// TIA Portal project "Practice" (V18)

(* hardware
DEVICE "S7-1500/ET200MP station_1"  S7-1500 station
   slot 0: "Rail_0"  Rack  6ES7 590-1***0-0AA0
   slot 1: "PLC_1"  CPU 1516F-3 PN/DP  6ES7 516-3FN01-0AB0  V2.1
      slot 3: "CPU display_1"  6ES7591-1BA00-0AA0
      slot 32768: "PROFINET interface_1"  X1
         slot 32769: "Port_1"  X1 P1
         slot 32770: "Port_2"  X1 P2
      slot 33024: "PROFINET interface_2"  X2
         slot 33025: "Port_1"  X2 P1
      slot 33280: "DP interface_1"  X3
   slot 2: "DI 16x24VDC HF_1"  DI 16x24VDC HF  6ES7 521-1BH00-0AB0  V2.2
   slot 3: "DQ 16x24VDC/0.5A HF_1"  DQ 16x24VDC/0.5A HF  6ES7 522-1BH01-0AB0  V1.1
   slot 4: "AI 8xU/I HF_1"  AI 8xU/I HF  6ES7 531-7NF00-0AB0  V1.2
   slot 5: "AQ 4xU/I HF_1"  AQ 4xU/I HF  6ES7 532-5ND00-0AB0  V1.1
*)

// ===== PLC "PLC_1"  CPU 1516F-3 PN/DP =====

VAR_GLOBAL   // PLC tag table "Default tag table"
   "ON" AT %I0.0 : Bool;
   "OFF" AT %I0.1 : Bool;
   "LAMP" AT %Q0.0 : Bool;
   "FAN" AT %Q0.1 : Bool;
   "WAR_LAMP" AT %Q0.2 : Bool;
   "CH_LP" AT %Q0.3 : Bool;
   "RST" AT %I0.2 : Bool;
   "POW_ON" AT %I0.3 : Bool;
   "CH_RST" AT %I0.4 : Bool;
   "CH_LAMP" AT %I0.5 : Bool;
END_VAR

DATA_BLOCK "Main_Safety_RTG1_DB"   // DB1, F_DB
{ S7_Optimized_Access := 'TRUE' }
NAME : FUSI
VERSION : 0.1
// stored: InstanceOfName Main_Safety_RTG1
"Main_Safety_RTG1"
BEGIN
END_DATA_BLOCK

DATA_BLOCK "SELF_HOLDING01_FB_DB"   // DB2
{ S7_Optimized_Access := 'TRUE' }
VERSION : 0.1
// stored: InstanceOfName SELF_HOLDING01_FB
"SELF_HOLDING01_FB"
BEGIN
END_DATA_BLOCK

DATA_BLOCK "SELF_HOLD_TIMER_FB02_DB"   // DB3
{ S7_Optimized_Access := 'TRUE' }
VERSION : 0.1
// stored: InstanceOfName SELF_HOLD_TIMER_FB02
"SELF_HOLD_TIMER_FB02"
BEGIN
END_DATA_BLOCK

DATA_BLOCK "SELF_HOLD_TOFF_FB03_DB"   // DB4
{ S7_Optimized_Access := 'TRUE' }
VERSION : 0.1
// stored: InstanceOfName SELF_HOLD_TOFF_FB03
"SELF_HOLD_TOFF_FB03"
BEGIN
END_DATA_BLOCK

DATA_BLOCK "LAMP_FAN_FLK_FB05_DB"   // DB5
{ S7_Optimized_Access := 'TRUE' }
VERSION : 0.1
// stored: InstanceOfName LAMP_FAN_FLK_FB05
"LAMP_FAN_FLK_FB05"
BEGIN
END_DATA_BLOCK

DATA_BLOCK "SELF_HOLD_RETENTIV_FB07_DB"   // DB6
{ S7_Optimized_Access := 'TRUE' }
VERSION : 0.1
// stored: InstanceOfName SELF_HOLD_RETENTIV_FB07
"SELF_HOLD_RETENTIV_FB07"
BEGIN
END_DATA_BLOCK

DATA_BLOCK "TOT_FUN_FB09_DB"   // DB7
{ S7_Optimized_Access := 'TRUE' }
VERSION : 0.1
// stored: InstanceOfName TOT_FUN_FB09
"TOT_FUN_FB09"
BEGIN
END_DATA_BLOCK

FUNCTION_BLOCK "Main_Safety_RTG1"   // FB1, F_FBD
{ S7_Optimized_Access := 'TRUE' }
BEGIN
END_FUNCTION_BLOCK

FUNCTION_BLOCK "SELF_HOLDING01_FB"   // FB2, LAD
TITLE = 자기유지 회로를 사용하여 램프 점등하기
{ S7_Optimized_Access := 'TRUE' }
VERSION : 0.1
   VAR_INPUT
      ON : Bool;
      OFF : Bool;
   END_VAR
   VAR_OUTPUT
      LAMP : Bool;
   END_VAR
   VAR
      K1 : Bool;
   END_VAR
BEGIN

REGION Network 1: 램프 점등을 위한 자기유지회로
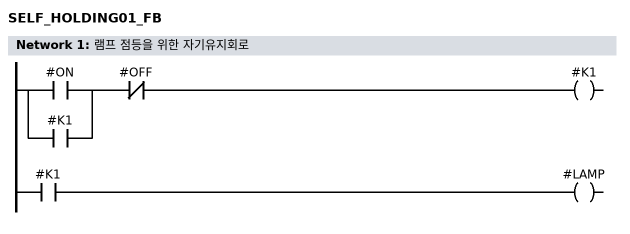
   RUNG wire#powerrail
      Contact( #ON )
      wire#w1
      I_Contact( #OFF )
      Coil( #K1 )
   END_RUNG
   RUNG wire#powerrail
      Contact( #K1 )
   END_RUNG wire#w1
   RUNG wire#powerrail
      Contact( #K1 )
      Coil( #LAMP )
   END_RUNG
   // the same network as SCL:
   #K1 := (#ON OR #K1) AND NOT #OFF;
   #LAMP := #K1;
END_REGION
END_FUNCTION_BLOCK

FUNCTION_BLOCK "SELF_HOLD_TIMER_FB02"   // FB3, LAD
TITLE = 자기유지 회로와 타이머의 조합 1
{ S7_Optimized_Access := 'TRUE' }
VERSION : 0.1
   VAR_INPUT
      ON : Bool;
      OFF : Bool;
   END_VAR
   VAR_OUTPUT
      LAMP : Bool;
      FAN : Bool;
   END_VAR
   VAR
      K1 : Bool;
      K2 : Bool;
      T1_Q : Bool;
      IEC_Timer_0_Instance : TON_TIME;
   END_VAR
BEGIN

REGION Network 1: 램프 제어 자기유지회로
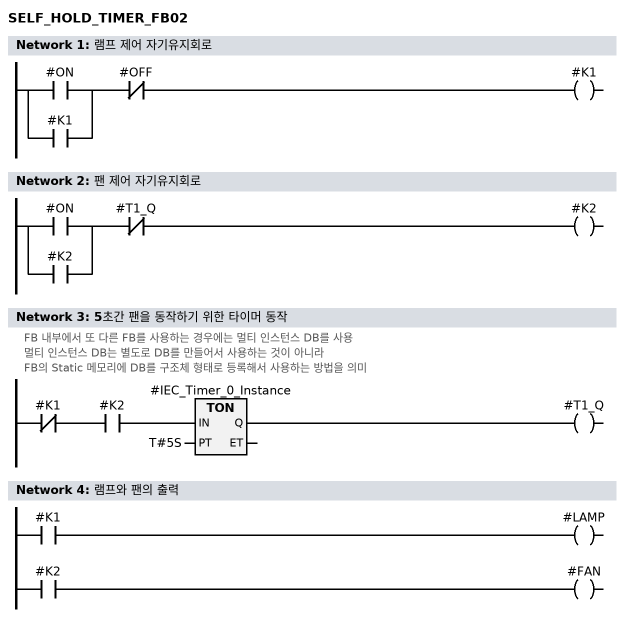
   RUNG wire#powerrail
      Contact( #ON )
      wire#w1
      I_Contact( #OFF )
      Coil( #K1 )
   END_RUNG
   RUNG wire#powerrail
      Contact( #K1 )
   END_RUNG wire#w1
   // the same network as SCL:
   #K1 := (#ON OR #K1) AND NOT #OFF;
END_REGION

REGION Network 2: 팬 제어 자기유지회로
   RUNG wire#powerrail
      Contact( #ON )
      wire#w1
      I_Contact( #T1_Q )
      Coil( #K2 )
   END_RUNG
   RUNG wire#powerrail
      Contact( #K2 )
   END_RUNG wire#w1
   // the same network as SCL:
   #K2 := (#ON OR #K2) AND NOT #T1_Q;
END_REGION

REGION Network 3: 5초간 팬을 동작하기 위한 타이머 동작
   // FB 내부에서 또 다른 FB를 사용하는 경우에는 멀티 인스턴스 DB를 사용
   // 
   // 멀티 인스턴스 DB는 별도로 DB를 만들어서 사용하는 것이 아니라
   // FB의 Static 메모리에 DB를 구조체 형태로 등록해서 사용하는 방법을 의미
   #IEC_Timer_0_Instance(IN := NOT #K1 AND #K2, PT := T#5S);   // TON
   #T1_Q := #IEC_Timer_0_Instance.Q;
END_REGION

REGION Network 4: 램프와 팬의 출력
   RUNG wire#powerrail
      Contact( #K1 )
      Coil( #LAMP )
   END_RUNG
   RUNG wire#powerrail
      Contact( #K2 )
      Coil( #FAN )
   END_RUNG
   // the same network as SCL:
   #LAMP := #K1;
   #FAN := #K2;
END_REGION
END_FUNCTION_BLOCK

FUNCTION_BLOCK "SELF_HOLD_TOFF_FB03"   // FB4, LAD
TITLE = 자기유지 회로와 타이머의 조합 2
{ S7_Optimized_Access := 'TRUE' }
VERSION : 0.1
   VAR_INPUT
      ON : Bool;
      OFF : Bool;
   END_VAR
   VAR_OUTPUT
      LAMP : Bool;
      FAN : Bool;
   END_VAR
   VAR
      K1 : Bool;
      K2 : Bool;
      IEC_Timer_0_Instance : TOF_TIME;
   END_VAR
BEGIN

REGION Network 1: 램프 제어 자기유지회로
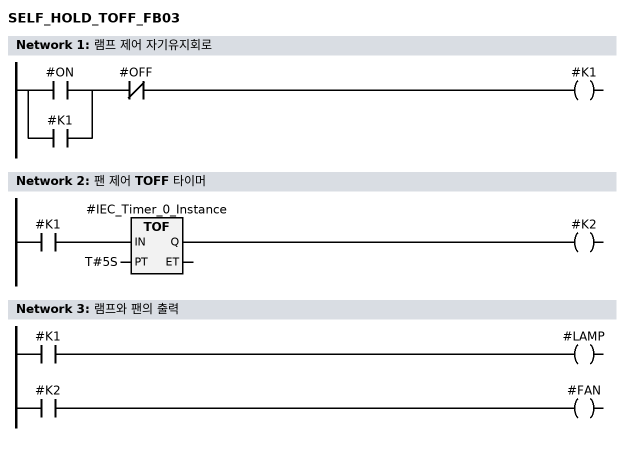
   RUNG wire#powerrail
      Contact( #ON )
      wire#w1
      I_Contact( #OFF )
      Coil( #K1 )
   END_RUNG
   RUNG wire#powerrail
      Contact( #K1 )
   END_RUNG wire#w1
   // the same network as SCL:
   #K1 := (#ON OR #K1) AND NOT #OFF;
END_REGION

REGION Network 2: 팬 제어 TOFF 타이머
   #IEC_Timer_0_Instance(IN := #K1, PT := T#5S);   // TOF
   #K2 := #IEC_Timer_0_Instance.Q;
END_REGION

REGION Network 3: 램프와 팬의 출력
   RUNG wire#powerrail
      Contact( #K1 )
      Coil( #LAMP )
   END_RUNG
   RUNG wire#powerrail
      Contact( #K2 )
      Coil( #FAN )
   END_RUNG
   // the same network as SCL:
   #LAMP := #K1;
   #FAN := #K2;
END_REGION
END_FUNCTION_BLOCK

FUNCTION_BLOCK "FLICKER_FB04"   // FB5, LAD
TITLE = 플리커 타이머 사용하기
{ S7_Optimized_Access := 'TRUE' }
VERSION : 0.1
   VAR_INPUT
      ON : Bool;
   END_VAR
   VAR_OUTPUT
      FLK_OUT : Bool;
   END_VAR
   VAR
      T1_Q : Bool;
      T1_ET : Time;
      IEC_Timer_0_Instance : TON_TIME;
   END_VAR
   VAR_TEMP   // added for the SCL form of the ladder/FBD networks
      _w1 : Bool;
   END_VAR
BEGIN

REGION Network 1: 1Hz주기를 가진 FLICKER 타이머
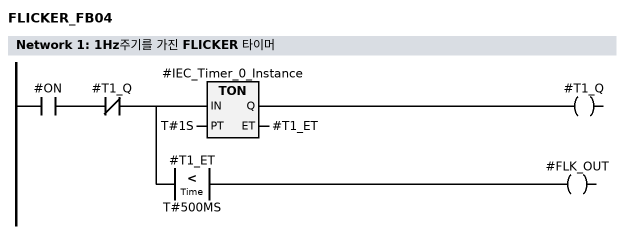
   #_w1 := #ON AND NOT #T1_Q;
   #IEC_Timer_0_Instance(IN := #_w1, PT := T#1S, ET => #T1_ET);   // TON
   #T1_Q := #IEC_Timer_0_Instance.Q;
   #FLK_OUT := #_w1 AND (#T1_ET < T#500MS);
END_REGION
END_FUNCTION_BLOCK

FUNCTION_BLOCK "LAMP_FAN_FLK_FB05"   // FB6, LAD
TITLE = 플리커 타이머 사용하기
{ S7_Optimized_Access := 'TRUE' }
VERSION : 0.1
   VAR_INPUT
      ON : Bool;
      OFF : Bool;
   END_VAR
   VAR_OUTPUT
      LAMP : Bool;
      FAN : Bool;
      WAR_LAMP : Bool;
   END_VAR
   VAR
      K1 : Bool;
      K2 : Bool;
      SELF_HOLD_TOFF_FB03_Instance : "SELF_HOLD_TOFF_FB03";
      FLICKER_FB04_Instance : "FLICKER_FB04";
   END_VAR
BEGIN

REGION Network 1: FB05에서 FB03 호출
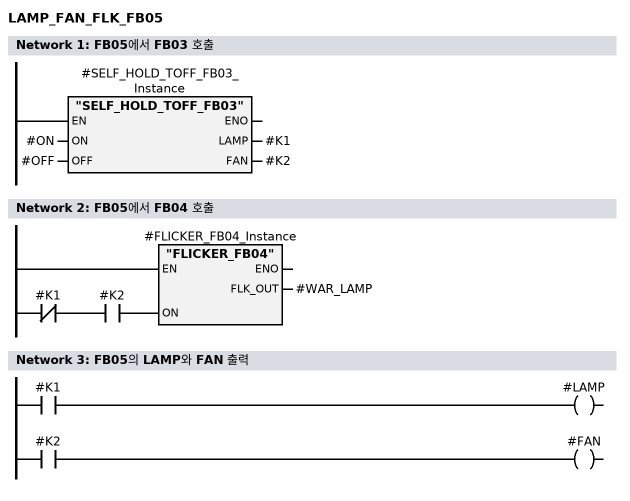
   RUNG wire#powerrail
      #SELF_HOLD_TOFF_FB03_Instance(ON := #ON, OFF := #OFF, LAMP => #K1, FAN => #K2)
   END_RUNG
   // the same network as SCL:
   #SELF_HOLD_TOFF_FB03_Instance(ON := #ON, OFF := #OFF, LAMP => #K1, FAN => #K2);   // "SELF_HOLD_TOFF_FB03"
END_REGION

REGION Network 2: FB05에서 FB04 호출
   RUNG wire#powerrail
      #FLICKER_FB04_Instance(ON := wire#w1, FLK_OUT => #WAR_LAMP)
   END_RUNG
   RUNG wire#powerrail
      I_Contact( #K1 )
      Contact( #K2 )
   END_RUNG wire#w1
   // the same network as SCL:
   #FLICKER_FB04_Instance(ON := NOT #K1 AND #K2, FLK_OUT => #WAR_LAMP);   // "FLICKER_FB04"
END_REGION

REGION Network 3: FB05의 LAMP와 FAN 출력
   RUNG wire#powerrail
      Contact( #K1 )
      Coil( #LAMP )
   END_RUNG
   RUNG wire#powerrail
      Contact( #K2 )
      Coil( #FAN )
   END_RUNG
   // the same network as SCL:
   #LAMP := #K1;
   #FAN := #K2;
END_REGION
END_FUNCTION_BLOCK

FUNCTION_BLOCK "RETENTIV_TIME_FB06"   // FB7, LAD
TITLE = PLC의 전원 ON/OFF에 관계없이 경과시간과 카운터의 값을 기억하기 위해서
{ S7_Optimized_Access := 'TRUE' }
VERSION : 0.1
   VAR_INPUT
      ON : Bool;
      RST : Bool;
   END_VAR
   VAR_OUTPUT
      OUT : Bool;
   END_VAR
   VAR
      T1_Q : Bool;
      C1_Q : Bool;
   END_VAR
   VAR RETAIN
      IEC_Timer_0_Instance : TONR_TIME;
      IEC_Counter_0_Instance : CTU_INT;
   END_VAR
BEGIN

REGION Network 1: 적산타이머의 동작
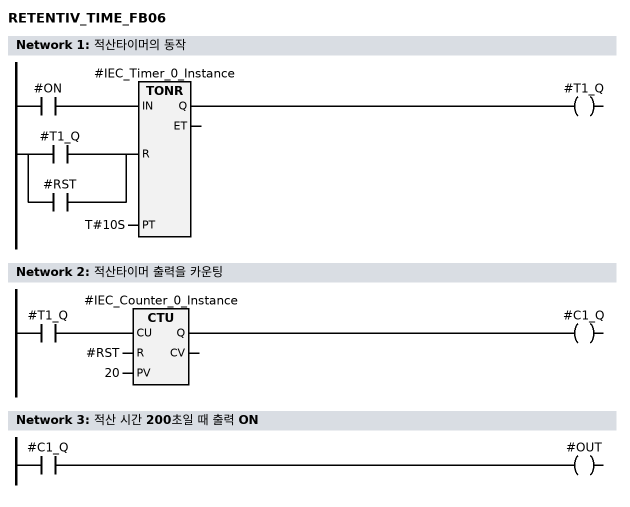
   #IEC_Timer_0_Instance(IN := #ON, R := #T1_Q OR #RST, PT := T#10S);   // TONR
   #T1_Q := #IEC_Timer_0_Instance.Q;
END_REGION

REGION Network 2: 적산타이머 출력을 카운팅
   #IEC_Counter_0_Instance(CU := #T1_Q, R := #RST, PV := 20);   // CTU
   #C1_Q := #IEC_Counter_0_Instance.Q;
END_REGION

REGION Network 3: 적산 시간 200초일 때 출력 ON
   RUNG wire#powerrail
      Contact( #C1_Q )
      Coil( #OUT )
   END_RUNG
   // the same network as SCL:
   #OUT := #C1_Q;
END_REGION
END_FUNCTION_BLOCK

FUNCTION_BLOCK "SELF_HOLD_RETENTIV_FB07"   // FB8, LAD
TITLE = FB1의 램프 출력은 FB6의 ON 입력으로 사용(K1 지정)
{ S7_Optimized_Access := 'TRUE' }
VERSION : 0.1
   VAR_INPUT
      ON : Bool;
      OFF : Bool;
      RST : Bool;
   END_VAR
   VAR_OUTPUT
      LAMP : Bool;
      CH_LP : Bool;
   END_VAR
   VAR
      K1 : Bool;
      SELF_HOLDING01_FB_Instance : "SELF_HOLDING01_FB";
      RETENTIV_TIME_FB06_Instance : "RETENTIV_TIME_FB06";
   END_VAR
BEGIN

REGION Network 1: 램프 점들을 위한 자기유지회로
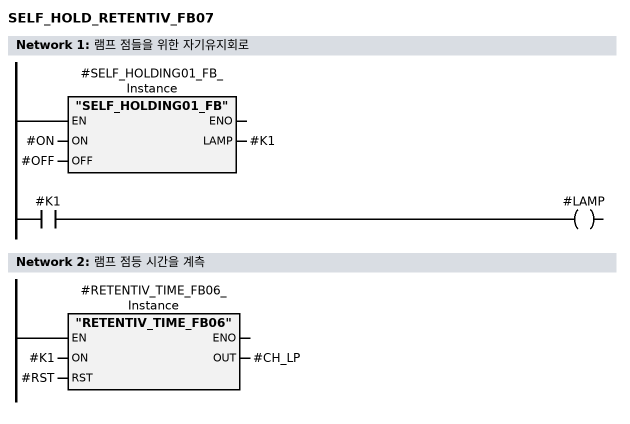
   RUNG wire#powerrail
      #SELF_HOLDING01_FB_Instance(ON := #ON, OFF := #OFF, LAMP => #K1)
   END_RUNG
   RUNG wire#powerrail
      Contact( #K1 )
      Coil( #LAMP )
   END_RUNG
   // the same network as SCL:
   #SELF_HOLDING01_FB_Instance(ON := #ON, OFF := #OFF, LAMP => #K1);   // "SELF_HOLDING01_FB"
   #LAMP := #K1;
END_REGION

REGION Network 2: 램프 점등 시간을 계측
   RUNG wire#powerrail
      #RETENTIV_TIME_FB06_Instance(ON := #K1, RST := #RST, OUT => #CH_LP)
   END_RUNG
   // the same network as SCL:
   #RETENTIV_TIME_FB06_Instance(ON := #K1, RST := #RST, OUT => #CH_LP);   // "RETENTIV_TIME_FB06"
END_REGION
END_FUNCTION_BLOCK

FUNCTION_BLOCK "FF_FUN_FB08"   // FB9, LAD
{ S7_Optimized_Access := 'TRUE' }
VERSION : 0.1
   VAR_INPUT
      ON_OFF : Bool;
      CH_RST : Bool;
   END_VAR
   VAR_OUTPUT
      ON_OUT : Bool;
      OFF_OUT : Bool;
      RST_OUT : Bool;
   END_VAR
   VAR
      K1 : Bool;
      K2 : Bool;
      R_EG01 : Bool;
      R_EG02 : Bool;
      F_EG01 : Bool;
      T1_Q : Bool;
      IEC_Timer_0_Instance : TON_TIME;
   END_VAR
BEGIN

REGION Network 1: 스위치 입력을 상승펄스 신호로 변경하여 K2를 토글 동작하도록 프로그램 작성
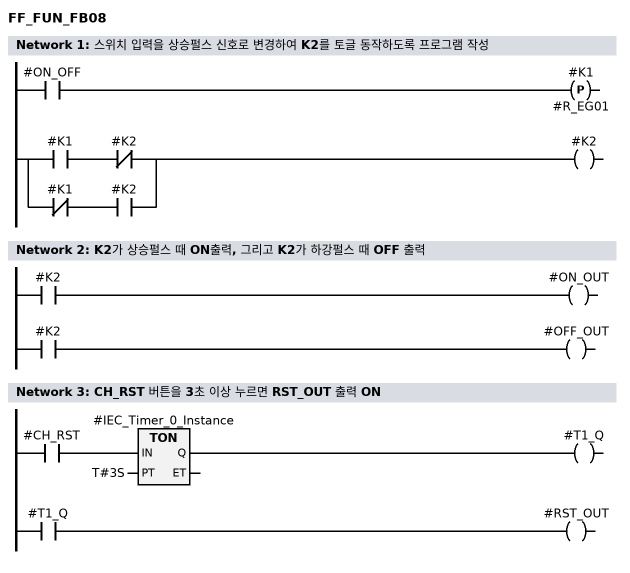
   #K1 := #ON_OFF AND NOT #R_EG01;   // rising edge
   #R_EG01 := #ON_OFF;
   #K2 := (#K1 AND NOT #K2) OR (NOT #K1 AND #K2);
END_REGION

REGION Network 2: K2가 상승펄스 때 ON출력, 그리고 K2가 하강펄스 때 OFF 출력
   RUNG wire#powerrail
      Contact( #K2 )
      Coil( #ON_OUT )
   END_RUNG
   RUNG wire#powerrail
      Contact( #K2 )
      Coil( #OFF_OUT )
   END_RUNG
   // the same network as SCL:
   #ON_OUT := #K2;
   #OFF_OUT := #K2;
END_REGION

REGION Network 3: CH_RST 버튼을 3초 이상 누르면 RST_OUT 출력 ON
   #IEC_Timer_0_Instance(IN := #CH_RST, PT := T#3S);   // TON
   #T1_Q := #IEC_Timer_0_Instance.Q;
   #RST_OUT := #T1_Q;
END_REGION
END_FUNCTION_BLOCK

FUNCTION_BLOCK "TOT_FUN_FB09"   // FB10, LAD
{ S7_Optimized_Access := 'TRUE' }
VERSION : 0.1
   VAR_INPUT
      POW_ON : Bool;
      CH_RST : Bool;
   END_VAR
   VAR_OUTPUT
      LAMP : Bool;
      FAN : Bool;
      WAR_LAMP : Bool;
      CH_LAMP : Bool;
   END_VAR
   VAR
      K1 : Bool;
      K2 : Bool;
      K3 : Bool;
      FF_FUN_FB08_Instance : "FF_FUN_FB08";
      LAMP_FAN_FLK_FB05_Instance : "LAMP_FAN_FLK_FB05";
      RETENTIV_TIME_FB06_Instance : "RETENTIV_TIME_FB06";
   END_VAR
BEGIN

REGION Network 1: 전원 버튼과 램프 교환 버튼 기능 구현
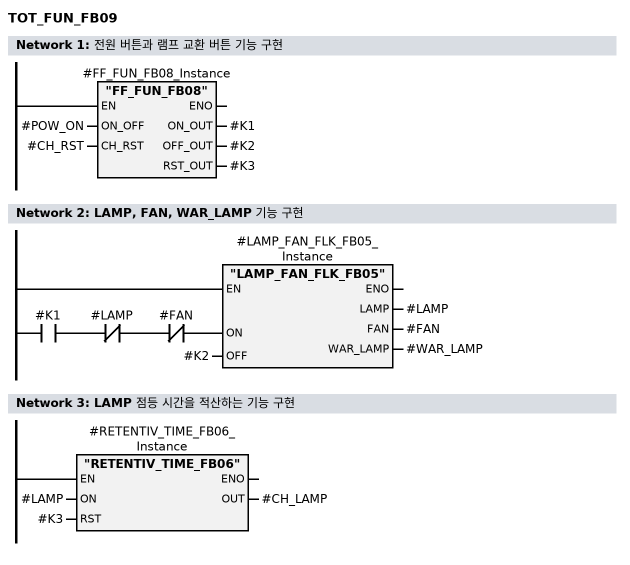
   RUNG wire#powerrail
      #FF_FUN_FB08_Instance(ON_OFF := #POW_ON, CH_RST := #CH_RST, ON_OUT => #K1, OFF_OUT => #K2, RST_OUT => #K3)
   END_RUNG
   // the same network as SCL:
   #FF_FUN_FB08_Instance(ON_OFF := #POW_ON, CH_RST := #CH_RST, ON_OUT => #K1, OFF_OUT => #K2, RST_OUT => #K3);   // "FF_FUN_FB08"
END_REGION

REGION Network 2: LAMP, FAN, WAR_LAMP 기능 구현
   RUNG wire#powerrail
      #LAMP_FAN_FLK_FB05_Instance(ON := wire#w1, OFF := #K2, LAMP => #LAMP, FAN => #FAN, WAR_LAMP => #WAR_LAMP)
   END_RUNG
   RUNG wire#powerrail
      Contact( #K1 )
      I_Contact( #LAMP )
      I_Contact( #FAN )
   END_RUNG wire#w1
   // the same network as SCL:
   #LAMP_FAN_FLK_FB05_Instance(ON := #K1 AND NOT #LAMP AND NOT #FAN,   // "LAMP_FAN_FLK_FB05"
                           OFF := #K2,
                           LAMP => #LAMP,
                           FAN => #FAN,
                           WAR_LAMP => #WAR_LAMP);
END_REGION

REGION Network 3: LAMP 점등 시간을 적산하는 기능 구현
   RUNG wire#powerrail
      #RETENTIV_TIME_FB06_Instance(ON := #LAMP, RST := #K3, OUT => #CH_LAMP)
   END_RUNG
   // the same network as SCL:
   #RETENTIV_TIME_FB06_Instance(ON := #LAMP, RST := #K3, OUT => #CH_LAMP);   // "RETENTIV_TIME_FB06"
END_REGION

REGION Network 4
   // ※ 경고 내용
   // 
   // tag is declared as an output and cannot be read
   // → 출력으로 지정된 태그를 입력으로 사용했다는 것
END_REGION
END_FUNCTION_BLOCK

FUNCTION_BLOCK "FF_FUN_BLK"   // FB100, LAD
{ S7_Optimized_Access := 'TRUE' }
VERSION : 0.1
// I0.0 : 전원
// I0.1 : 교환/리셋
// Q0.0 : 램프
// Q0.1 : 팬
// Q0.2 : 경고등
// Q0.3 : 램프 교환
   VAR_INPUT
      ON : Bool;
   END_VAR
   VAR_OUTPUT
      OUT : Bool;
   END_VAR
   VAR
      PLS_SIG : Bool;
      K1 : Bool;
      R_EG01 : Bool;
   END_VAR
BEGIN

REGION Network 1: ON입력 신호를 상승펄스 출력으로 처리
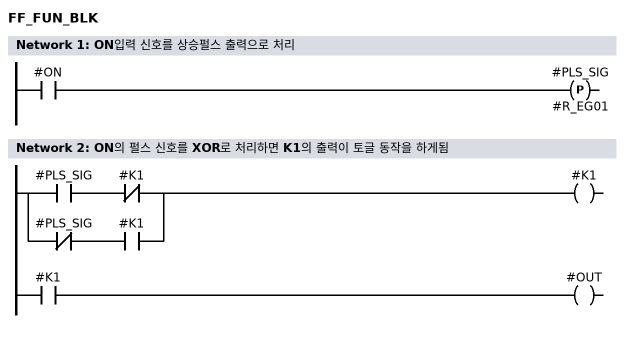
   #PLS_SIG := #ON AND NOT #R_EG01;   // rising edge
   #R_EG01 := #ON;
END_REGION

REGION Network 2: ON의 펄스 신호를 XOR로 처리하면 K1의 출력이 토글 동작을 하게됨
   RUNG wire#powerrail
      Contact( #PLS_SIG )
      I_Contact( #K1 )
      wire#w1
      Coil( #K1 )
   END_RUNG
   RUNG wire#powerrail
      I_Contact( #PLS_SIG )
      Contact( #K1 )
   END_RUNG wire#w1
   RUNG wire#powerrail
      Contact( #K1 )
      Coil( #OUT )
   END_RUNG
   // the same network as SCL:
   #K1 := (#PLS_SIG AND NOT #K1) OR (NOT #PLS_SIG AND #K1);
   #OUT := #K1;
END_REGION
END_FUNCTION_BLOCK

FUNCTION_BLOCK "FF_TIMER_BLK"   // FB101, LAD
{ S7_Optimized_Access := 'TRUE' }
VERSION : 0.1
   VAR_INPUT
      ON : Bool;
   END_VAR
   VAR_OUTPUT
      FF_OUT : Bool;
   END_VAR
   VAR
      T1_Q : Bool;
      IEC_Timer_0_Instance : TON_TIME;
      FF_FUN_BLK_Instance : "FF_FUN_BLK";
   END_VAR
BEGIN

REGION Network 1: ON 버튼이 3초 이상 눌러진 것을 검출하기 위해 TON 사용
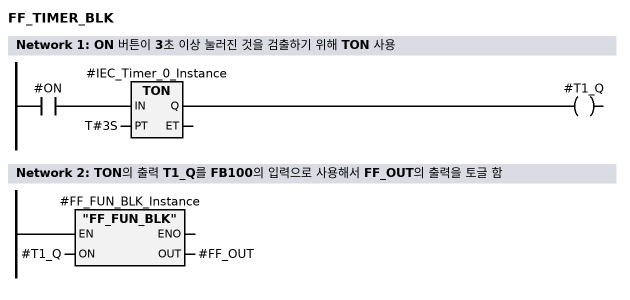
   #IEC_Timer_0_Instance(IN := #ON, PT := T#3S);   // TON
   #T1_Q := #IEC_Timer_0_Instance.Q;
END_REGION

REGION Network 2: TON의 출력 T1_Q를 FB100의 입력으로 사용해서 FF_OUT의 출력을 토글 함
   RUNG wire#powerrail
      #FF_FUN_BLK_Instance(ON := #T1_Q, OUT => #FF_OUT)
   END_RUNG
   // the same network as SCL:
   #FF_FUN_BLK_Instance(ON := #T1_Q, OUT => #FF_OUT);   // "FF_FUN_BLK"
END_REGION
END_FUNCTION_BLOCK

ORGANIZATION_BLOCK "Main"   // OB1, LAD, ProgramCycle
TITLE = "Main Program Sweep (Cycle)"
{ S7_Optimized_Access := 'TRUE' }
VERSION : 0.1
   VAR_INPUT
      Initial_Call : Bool;   // Initial call of this OB
      Remanence : Bool;   // =True, if remanent data are available
   END_VAR
BEGIN

REGION Network 1: Practice_1
   // 램프 점등을 위한 자기유지회로
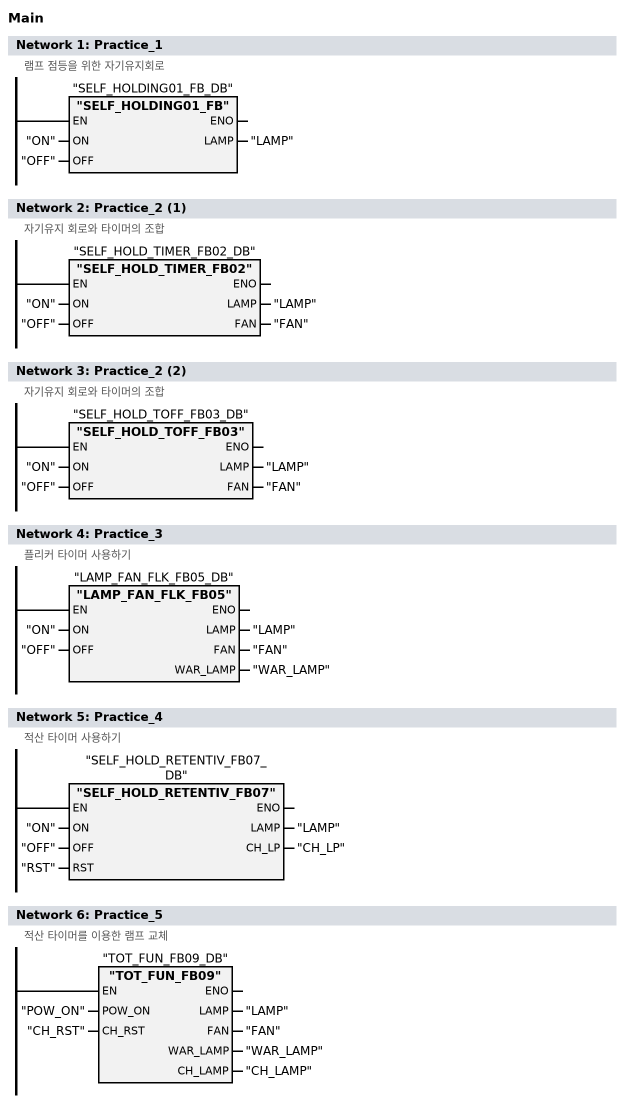
   RUNG wire#powerrail
      "SELF_HOLDING01_FB_DB"(ON := "ON", OFF := "OFF", LAMP => "LAMP")
   END_RUNG
   // the same network as SCL:
   "SELF_HOLDING01_FB_DB"(ON := "ON", OFF := "OFF", LAMP => "LAMP");   // "SELF_HOLDING01_FB"
END_REGION

REGION Network 2: Practice_2 (1)
   // 자기유지 회로와 타이머의 조합
   RUNG wire#powerrail
      "SELF_HOLD_TIMER_FB02_DB"(ON := "ON", OFF := "OFF", LAMP => "LAMP", FAN => "FAN")
   END_RUNG
   // the same network as SCL:
   "SELF_HOLD_TIMER_FB02_DB"(ON := "ON", OFF := "OFF", LAMP => "LAMP", FAN => "FAN");   // "SELF_HOLD_TIMER_FB02"
END_REGION

REGION Network 3: Practice_2 (2)
   // 자기유지 회로와 타이머의 조합
   RUNG wire#powerrail
      "SELF_HOLD_TOFF_FB03_DB"(ON := "ON", OFF := "OFF", LAMP => "LAMP", FAN => "FAN")
   END_RUNG
   // the same network as SCL:
   "SELF_HOLD_TOFF_FB03_DB"(ON := "ON", OFF := "OFF", LAMP => "LAMP", FAN => "FAN");   // "SELF_HOLD_TOFF_FB03"
END_REGION

REGION Network 4: Practice_3
   // 플리커 타이머 사용하기
   RUNG wire#powerrail
      "LAMP_FAN_FLK_FB05_DB"(ON := "ON", OFF := "OFF", LAMP => "LAMP", FAN => "FAN", WAR_LAMP => "WAR_LAMP")
   END_RUNG
   // the same network as SCL:
   "LAMP_FAN_FLK_FB05_DB"(ON := "ON", OFF := "OFF", LAMP => "LAMP", FAN => "FAN", WAR_LAMP => "WAR_LAMP");   // "LAMP_FAN_FLK_FB05"
END_REGION

REGION Network 5: Practice_4
   // 적산 타이머 사용하기
   RUNG wire#powerrail
      "SELF_HOLD_RETENTIV_FB07_DB"(ON := "ON", OFF := "OFF", RST := "RST", LAMP => "LAMP", CH_LP => "CH_LP")
   END_RUNG
   // the same network as SCL:
   "SELF_HOLD_RETENTIV_FB07_DB"(ON := "ON", OFF := "OFF", RST := "RST", LAMP => "LAMP", CH_LP => "CH_LP");   // "SELF_HOLD_RETENTIV_FB07"
END_REGION

REGION Network 6: Practice_5
   // 적산 타이머를 이용한 램프 교체
   RUNG wire#powerrail
      "TOT_FUN_FB09_DB"(POW_ON := "POW_ON", CH_RST := "CH_RST", LAMP => "LAMP", FAN => "FAN", WAR_LAMP => "WAR_LAMP", CH_LAMP => "CH_LAMP")
   END_RUNG
   // the same network as SCL:
   "TOT_FUN_FB09_DB"(POW_ON := "POW_ON",   // "TOT_FUN_FB09"
                     CH_RST := "CH_RST",
                     LAMP => "LAMP",
                     FAN => "FAN",
                     WAR_LAMP => "WAR_LAMP",
                     CH_LAMP => "CH_LAMP");
END_REGION
END_ORGANIZATION_BLOCK